PROGRAM PRG_TEST
VAR
END_VAR

END_PROGRAM

(* stored: Version 1.1.0.1, ProductVersion 3.1.4024.12
   POU PRG_TEST: Id {426a6bfe-44e0-00d4-3713-2ee15ce3853f}, SpecialFunc None *)
